INTERFACE I_Queue

(* Removes element from the front of the queue. *)
METHOD Dequeue : T_DATA_TYPE
VAR_INPUT
END_VAR
END_METHOD

(* Empties/Clears/Deletes all elements on the stack. *)
METHOD Empty
END_METHOD

(* Adds element to the rear of the queue. *)
METHOD Enqueue
VAR_INPUT
	Data 	: T_DATA_TYPE;
END_VAR
END_METHOD

METHOD FB_exit : BOOL
VAR_INPUT
	bInCopyCode : BOOL; // if TRUE, the exit method is called for exiting an instance that is copied afterwards (online change).
END_VAR
END_METHOD

METHOD FB_init : BOOL
VAR_INPUT
	bInitRetains : BOOL; // if TRUE, the retain variables are initialized (warm start / cold start)
	bInCopyCode : BOOL;  // if TRUE, the instance afterwards gets moved into the copy code (online change)
END_VAR
END_METHOD

(* Checks of queue is empty. *)
METHOD Is_Empty : BOOL
VAR_INPUT
END_VAR
END_METHOD

// Gets element at any position of the queue, without removing it.
METHOD Peek : T_DATA_TYPE
VAR_INPUT
	nPosition : DINT;
END_VAR
END_METHOD

(* Traverse the queue and display each element as an array. *)
METHOD Show
VAR_IN_OUT
	aList : ARRAY[*] OF T_DATA_TYPE; // Array to display data in list.
END_VAR
END_METHOD

(* Gets size of the queue. *)
METHOD Size : DINT;
END_METHOD

END_INTERFACE

(* stored: Version 1.1.0.1, ProductVersion 3.1.4024.4
   Itf I_Queue: Id {88dc387d-7152-4d4a-bee6-f1274bfb5237}
   Method Dequeue: Id {04f7b95a-266f-4895-b766-645c7fd6c23c}
   Method Empty: Id {650a0080-6c1d-4b5e-9088-afcc874848bd}
   Method Enqueue: Id {e8a11593-9787-420f-ad5d-1568e96cecb2}
   Method FB_exit: Id {1174579a-395f-45f8-864e-c3b3d4e9333f}
   Method FB_init: Id {0bfd7fb0-2374-4bcb-87e0-26f0d0674b75}
   Method Is_Empty: Id {f8a89ecc-2bf3-4966-b6da-f5f1e59d45b8}
   Method Peek: Id {183439c7-78c9-44ff-abf1-e1d90c767ce6}
   Method Show: Id {8e00b43a-914a-45bf-8bc9-1d45764f6cb9}
   Method Size: Id {4595053a-2e27-4879-a5cf-3bc815c1966e} *)
